(* IEC 61131-3 sources: repolevel_ST_code_completion/output/0122完整版本_无planner目前sota/repoeval_ProductionLine/readful_result_no_provide, 5 files *)

(* ---- Motor_ResetFault.st ---- *)
VAR
	ResetDetect: r_trig;
END_VAR

ResetDetect(CLK := MotorI.FaultReset);

IF ResetDetect.Q THEN
	MotorO.FaultStatus := FALSE;
END_IF

RETURN;
END_OTHER

(* ---- Motor_SetFault.st ---- *)
VAR
	WaitTimer:TON;
	InternalSequenceDelay:TIME;
END_VAR

IF MotorI.Overload THEN
	MotorO.FaultStatus := TRUE;
	MotorO.Coil := FALSE;
END_IF;
RETURN;
END_OTHER

(* ---- Motor_SetWaitTime.st ---- *)
VAR
	WaitTimer:TON;
	InternalSequenceDelay:TIME;
END_VAR

InternalSequenceDelay := SequenceDelay;

IF MotorO.FaultStatus = FALSE THEN
	WaitTimer(IN := TRUE, PT := InternalSequenceDelay);
END_IF

IF WaitTimer.Q THEN
	MotorO.Coil := TRUE;
	WaitTimer(IN := FALSE);
	RETURN := TRUE;
ELSE
	RETURN := FALSE;
END_IF
END_OTHER

(* ---- Motor_TurnOff.st ---- *)
VAR
	WaitTimer:TON;
	InternalSequenceDelay:TIME;
END_VAR

MotorO.Coil := FALSE;
RETURN;
END_OTHER

(* ---- Motor_TurnOn.st ---- *)
VAR
	WaitTimer:TON;
	InternalSequenceDelay:TIME;
END_VAR

IF MotorO.FaultStatus = FALSE THEN
	WaitTimer(IN := TRUE, PT := InternalSequenceDelay);
END_IF

IF WaitTimer.Q THEN
	MotorO.Coil := TRUE;
	WaitTimer(IN := FALSE);
END_IF

RETURN;
END_OTHER
